(* Schneider Machine Expert - Basic project driveAPIREV3, file version 2.7.0.0 *)
(* ProjectInformations: Name=PlanPAS 2.0 *)

HARDWARE
  Cpu 0: TM221CE16T
  EthernetConfiguration: NetworkName=M221, IpAllocationMode=FixedAddress, IpAddress=192.168.0.2, SubnetMask=255.255.255.0
  SerialLineConfiguration: Baud=Baud19200, Parity=ParityEven, DataBits=DataBits8, StopBits=StopBits1, PhysicalMedium=PhysicalMediumRs485, TransmissionMode=TransmissionModeModbusRtu, SlaveId=1, Addressing=SlaveAddressing
  MastTask: UsePeriodScanMode=false, PeriodScan=100
  FastTask: Period=255
  CpuBehavior: StartingMode=StartAsPreviousState, AutoSaveRamOnEeprom=true, WatchdogPeriod=250

SYMBOLS  (address, symbol, comment, settings)
  %M0         "ESTEIRA"
  %M1         "AVANÇA PISTÃO 1"
  %M2         "AVANÇA PISTÃO 2"
  %M3         "AVANÇA PISTÃO 3"
  %M4         "RETORNA PISTÃO 3"
  %M5         "IDENTIFICA PEÇA NA ESTEIRA (CAPACITIVO)"
  %M6         "LIMPA AVISOS"
  %M10        "MEDIA"
  %M11        "GRANDE"
  %M12        "METAL"
  %M14        "CHEGADA DE PEÇA BOX 2"
  %M15        "CHEGADA DE PEÇA BOX 1"
  %M16        "CHEGADA DE PEÇA BOX 3"
  %M17        "CHEGADA DE PEÇA BOX 4"
  %M20        "PEQ_NMET"
  %M21        "PEQ_MET"
  %M22        "MED_NMET"
  %M23        "MED_MET"
  %M24        "GRD_NMET"
  %M25        "GRD_MET"
  %M30      INICIAR
  %M31      PARAR
  %M32      REPROG
  %M33      VOLTAR
  %M34      INICIADO
  %M40        "INICIAR AUX"
  %M41        "PARAR AUX"
  %M42        "REPROGRAMAR AUX"
  %M43        "VOLTAR AUX"
  %M44        "ZERA MEMORIA SOLICITAÇÕES"
  %MW0        "AVISOS"
  %MW10     CX1MG  "SOLICITAÇÃO"
  %MW11     CX1MM
  %MW12     CX1MP
  %MW13     CX1NMG
  %MW14     CX1NMM
  %MW15     CX1NMP
  %MW16     CX2MG
  %MW17     CX2MM
  %MW18     CX2MP
  %MW19     CX2NMG
  %MW20     CX2NMM
  %MW21     CX2NMP
  %MW22     CX3MG
  %MW23     CX3MM
  %MW24     CX3MP
  %MW25     CX3NMG
  %MW26     CX3NMM
  %MW27     CX3NMP
  %I0.0       "SENS_OTICO_MED"
  %I0.1       "SENS_OTICO_GDE"
  %I0.2       "SENS_INDUTIVO"
  %I0.3       "SENS_CAPACITIVO"
  %I0.4       "FC2"
  %I0.5       "FC1"
  %I0.6       "FC3"
  %I0.7       "FC4"
  %Q0.0       "M1"
  %Q0.1       "AP1"
  %Q0.2       "AP2"
  %Q0.3       "AP3"
  %Q0.5       "RP3"

POU Novo POU
  (* SectionNumber=1 *)

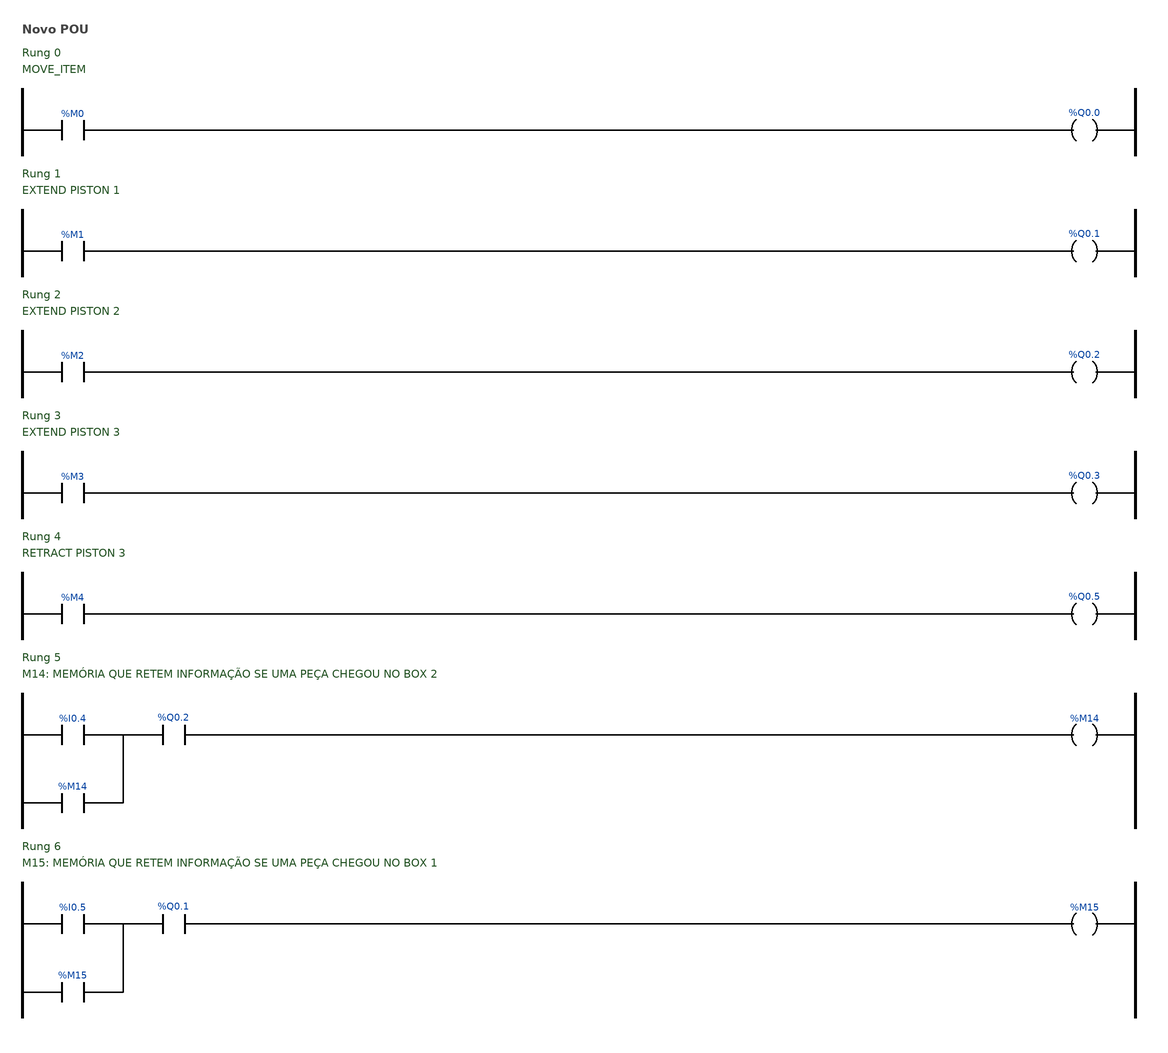

// Rung 0
// MOVE_ITEM
  LD %M0
  ST %Q0.0
  // as ST:
  //   %Q0.0 := %M0;

// Rung 1
// EXTEND PISTON 1
  LD %M1
  ST %Q0.1
  // as ST:
  //   %Q0.1 := %M1;

// Rung 2
// EXTEND PISTON 2
  LD %M2
  ST %Q0.2
  // as ST:
  //   %Q0.2 := %M2;

// Rung 3
// EXTEND PISTON 3
  LD %M3
  ST %Q0.3
  // as ST:
  //   %Q0.3 := %M3;

// Rung 4
// RETRACT PISTON 3
  LD %M4
  ST %Q0.5
  // as ST:
  //   %Q0.5 := %M4;

// Rung 5
// M14: MEMÓRIA QUE RETEM INFORMAÇÃO SE UMA PEÇA CHEGOU NO BOX 2
  LD %I0.4
  OR %M14
  AND %Q0.2
  ST %M14
  // as ST:
  //   %M14 := (%I0.4 OR %M14) AND %Q0.2;

// Rung 6
// M15: MEMÓRIA QUE RETEM INFORMAÇÃO SE UMA PEÇA CHEGOU NO BOX 1
  LD %I0.5
  OR %M15
  AND %Q0.1
  ST %M15
  // as ST:
  //   %M15 := (%I0.5 OR %M15) AND %Q0.1;

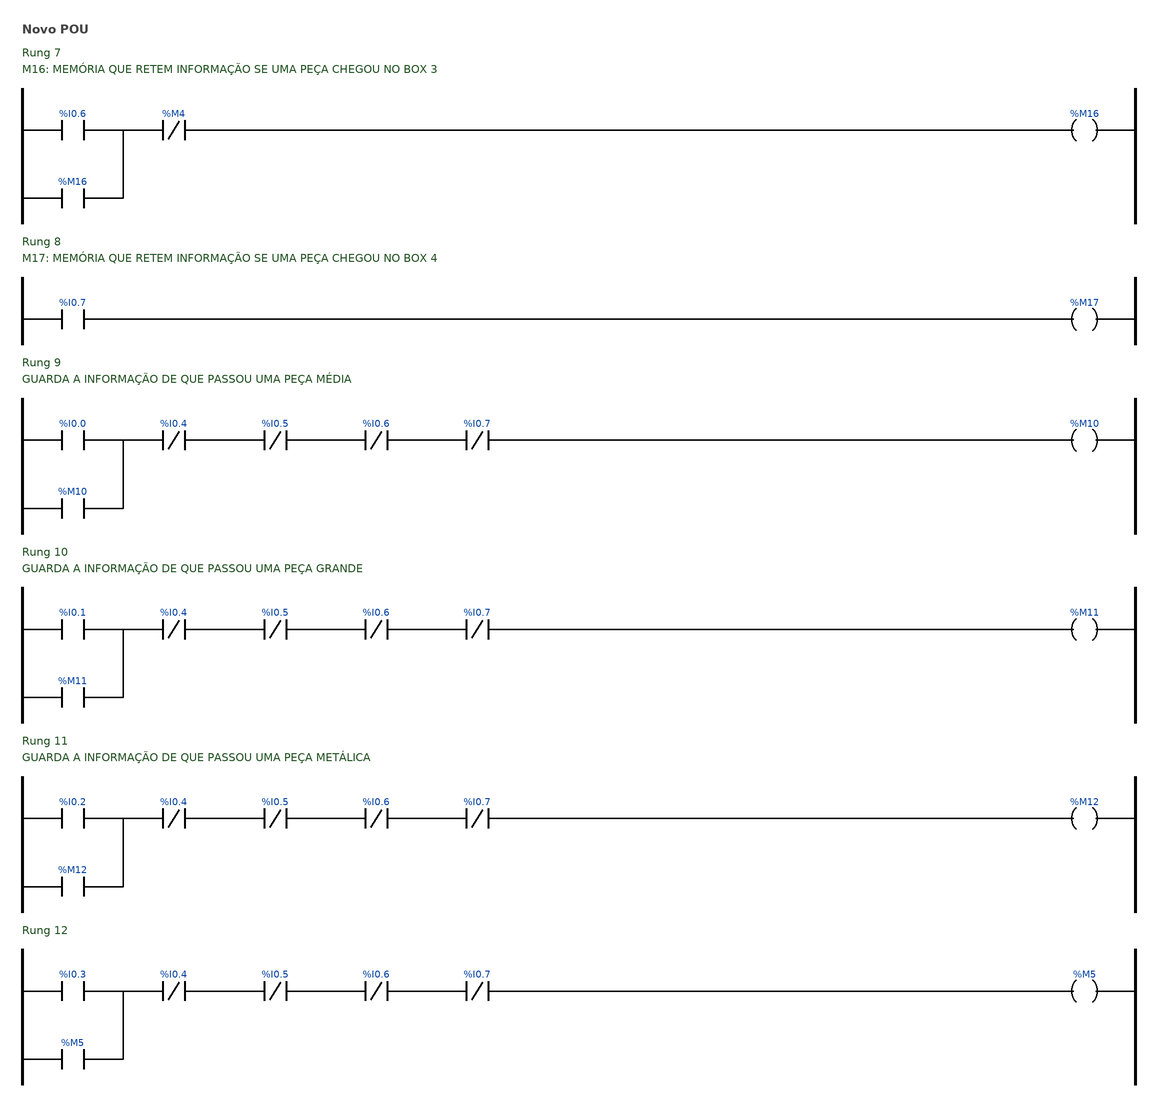

// Rung 7
// M16: MEMÓRIA QUE RETEM INFORMAÇÃO SE UMA PEÇA CHEGOU NO BOX 3
  LD %I0.6
  OR %M16
  ANDN %M4
  ST %M16
  // as ST:
  //   %M16 := (%I0.6 OR %M16) AND NOT %M4;

// Rung 8
// M17: MEMÓRIA QUE RETEM INFORMAÇÃO SE UMA PEÇA CHEGOU NO BOX 4
  LD %I0.7
  ST %M17
  // as ST:
  //   %M17 := %I0.7;

// Rung 9
// GUARDA A INFORMAÇÃO DE QUE PASSOU UMA PEÇA MÉDIA
  LD %I0.0
  OR %M10
  ANDN %I0.4
  ANDN %I0.5
  ANDN %I0.6
  ANDN %I0.7
  ST %M10
  // as ST:
  //   %M10 := (%I0.0 OR %M10) AND NOT %I0.4 AND NOT %I0.5 AND NOT %I0.6 AND NOT %I0.7;

// Rung 10
// GUARDA A INFORMAÇÃO DE QUE PASSOU UMA PEÇA GRANDE
  LD %I0.1
  OR %M11
  ANDN %I0.4
  ANDN %I0.5
  ANDN %I0.6
  ANDN %I0.7
  ST %M11
  // as ST:
  //   %M11 := (%I0.1 OR %M11) AND NOT %I0.4 AND NOT %I0.5 AND NOT %I0.6 AND NOT %I0.7;

// Rung 11
// GUARDA A INFORMAÇÃO DE QUE PASSOU UMA PEÇA METÁLICA
  LD %I0.2
  OR %M12
  ANDN %I0.4
  ANDN %I0.5
  ANDN %I0.6
  ANDN %I0.7
  ST %M12
  // as ST:
  //   %M12 := (%I0.2 OR %M12) AND NOT %I0.4 AND NOT %I0.5 AND NOT %I0.6 AND NOT %I0.7;

// Rung 12
  LD %I0.3
  OR %M5
  ANDN %I0.4
  ANDN %I0.5
  ANDN %I0.6
  ANDN %I0.7
  ST %M5
  // as ST:
  //   %M5 := (%I0.3 OR %M5) AND NOT %I0.4 AND NOT %I0.5 AND NOT %I0.6 AND NOT %I0.7;

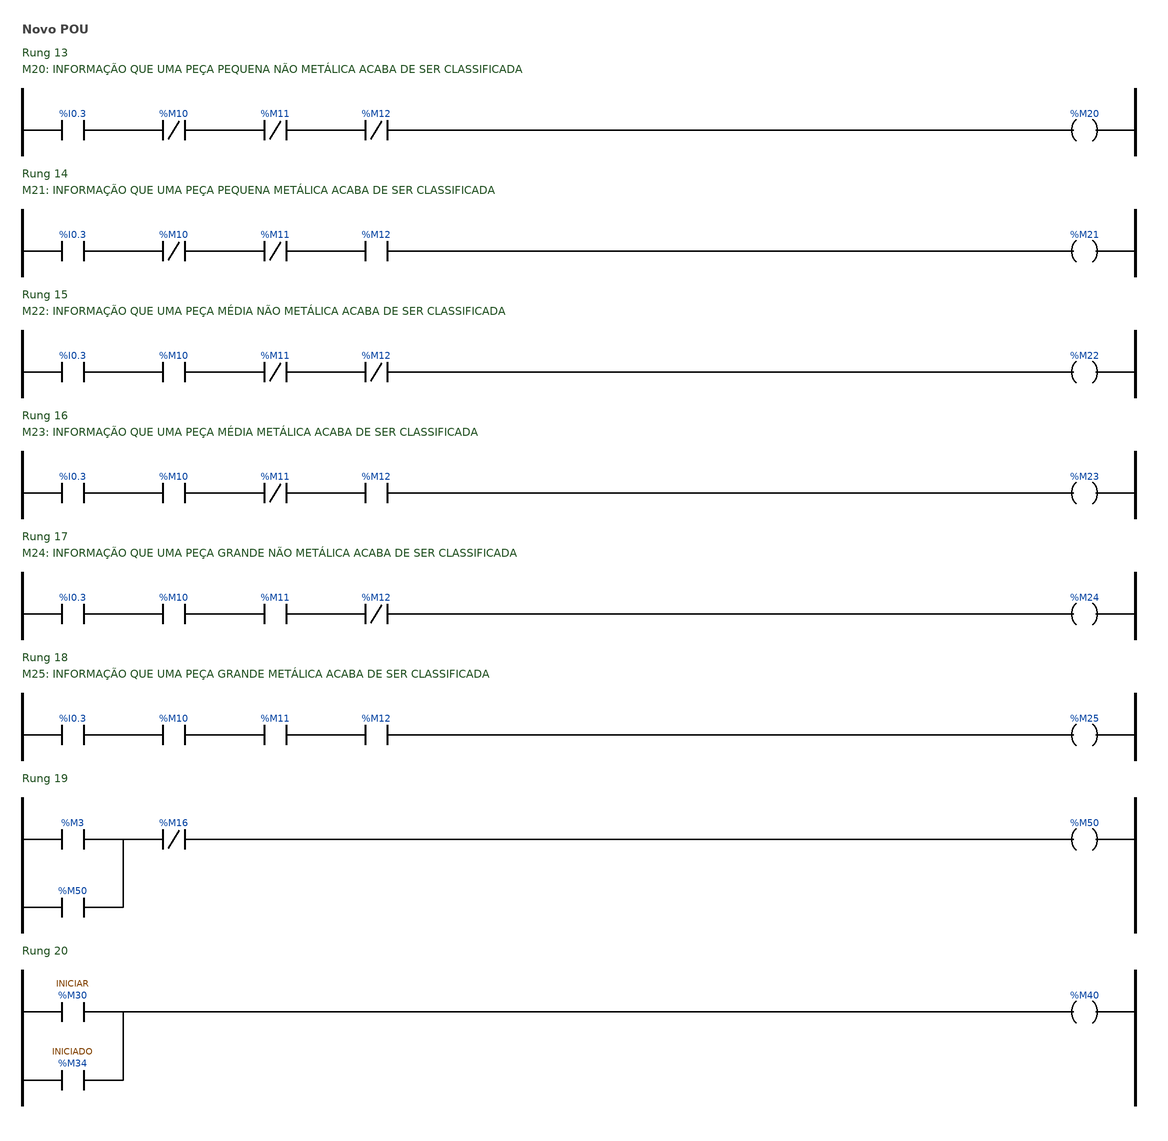

// Rung 13
// M20: INFORMAÇÃO QUE UMA PEÇA PEQUENA NÃO METÁLICA ACABA DE SER CLASSIFICADA
  LD %I0.3
  ANDN %M10
  ANDN %M11
  ANDN %M12
  ST %M20
  // as ST:
  //   %M20 := %I0.3 AND NOT %M10 AND NOT %M11 AND NOT %M12;

// Rung 14
// M21: INFORMAÇÃO QUE UMA PEÇA PEQUENA METÁLICA ACABA DE SER CLASSIFICADA
  LD %I0.3
  ANDN %M10
  ANDN %M11
  AND %M12
  ST %M21
  // as ST:
  //   %M21 := %I0.3 AND NOT %M10 AND NOT %M11 AND %M12;

// Rung 15
// M22: INFORMAÇÃO QUE UMA PEÇA MÉDIA NÃO METÁLICA ACABA DE SER CLASSIFICADA
  LD %I0.3
  AND %M10
  ANDN %M11
  ANDN %M12
  ST %M22
  // as ST:
  //   %M22 := %I0.3 AND %M10 AND NOT %M11 AND NOT %M12;

// Rung 16
// M23: INFORMAÇÃO QUE UMA PEÇA MÉDIA METÁLICA ACABA DE SER CLASSIFICADA
  LD %I0.3
  AND %M10
  ANDN %M11
  AND %M12
  ST %M23
  // as ST:
  //   %M23 := %I0.3 AND %M10 AND NOT %M11 AND %M12;

// Rung 17
// M24: INFORMAÇÃO QUE UMA PEÇA GRANDE NÃO METÁLICA ACABA DE SER CLASSIFICADA
  LD %I0.3
  AND %M10
  AND %M11
  ANDN %M12
  ST %M24
  // as ST:
  //   %M24 := %I0.3 AND %M10 AND %M11 AND NOT %M12;

// Rung 18
// M25: INFORMAÇÃO QUE UMA PEÇA GRANDE METÁLICA ACABA DE SER CLASSIFICADA
  LD %I0.3
  AND %M10
  AND %M11
  AND %M12
  ST %M25
  // as ST:
  //   %M25 := %I0.3 AND %M10 AND %M11 AND %M12;

// Rung 19
  LD %M3
  OR %M50
  ANDN %M16
  ST %M50
  // as ST:
  //   %M50 := (%M3 OR %M50) AND NOT %M16;

// Rung 20
  LD %M30                 (* INICIAR *)
  OR %M34                 (* INICIADO *)
  ST %M40
  // as ST:
  //   %M40 := INICIAR OR INICIADO;

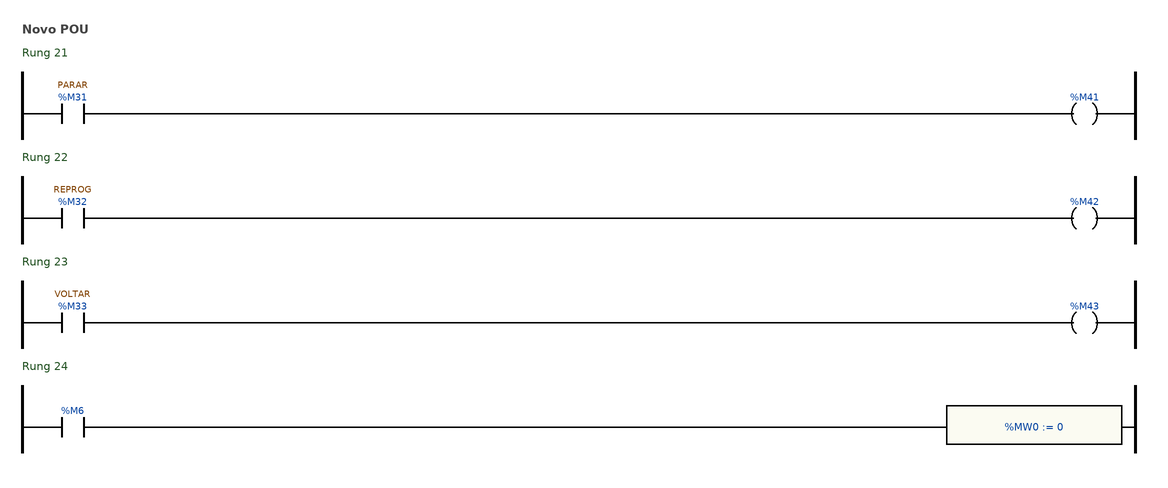

// Rung 21
  LD %M31                 (* PARAR *)
  ST %M41
  // as ST:
  //   %M41 := PARAR;

// Rung 22
  LD %M32                 (* REPROG *)
  ST %M42
  // as ST:
  //   %M42 := REPROG;

// Rung 23
  LD %M33                 (* VOLTAR *)
  ST %M43
  // as ST:
  //   %M43 := VOLTAR;

// Rung 24
  LD %M6
  [ %MW0 := 0 ]
  // as ST:
  //   IF %M6 THEN %MW0 := 0; END_IF;

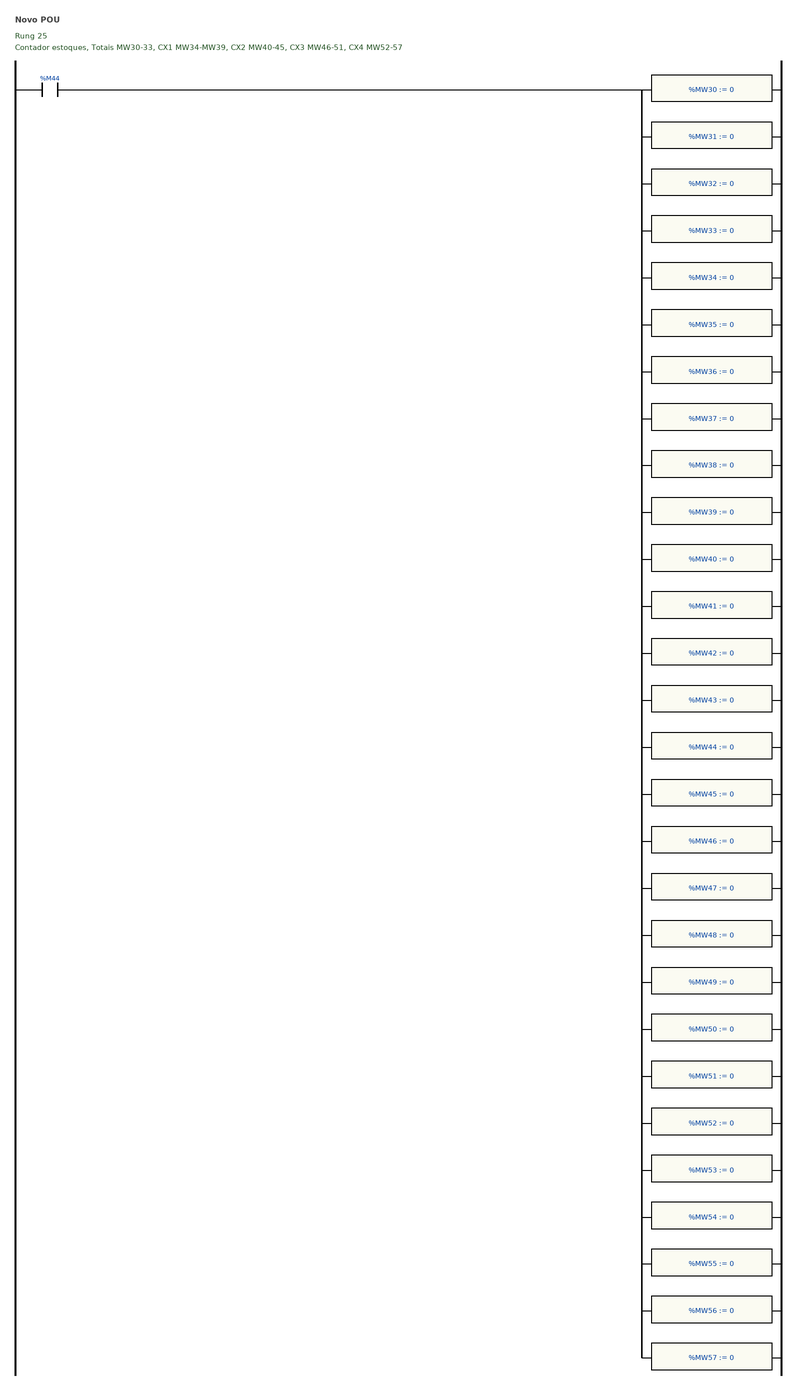

// Rung 25
// Contador estoques, Totais MW30-33, CX1 MW34-MW39, CX2 MW40-45, CX3 MW46-51, CX4 MW52-57
  LD %M44
  [ %MW30 := 0 ]
  [ %MW31 := 0 ]
  [ %MW32 := 0 ]
  [ %MW33 := 0 ]
  [ %MW34 := 0 ]
  [ %MW35 := 0 ]
  [ %MW36 := 0 ]
  [ %MW37 := 0 ]
  [ %MW38 := 0 ]
  [ %MW39 := 0 ]
  [ %MW40 := 0 ]
  [ %MW41 := 0 ]
  [ %MW42 := 0 ]
  [ %MW43 := 0 ]
  [ %MW44 := 0 ]
  [ %MW45 := 0 ]
  [ %MW46 := 0 ]
  [ %MW47 := 0 ]
  [ %MW48 := 0 ]
  [ %MW49 := 0 ]
  [ %MW50 := 0 ]
  [ %MW51 := 0 ]
  [ %MW52 := 0 ]
  [ %MW53 := 0 ]
  [ %MW54 := 0 ]
  [ %MW55 := 0 ]
  [ %MW56 := 0 ]
  [ %MW57 := 0 ]
  // as ST:
  //   IF %M44 THEN %MW30 := 0; END_IF;
  //   IF %M44 THEN %MW31 := 0; END_IF;
  //   IF %M44 THEN %MW32 := 0; END_IF;
  //   IF %M44 THEN %MW33 := 0; END_IF;
  //   IF %M44 THEN %MW34 := 0; END_IF;
  //   IF %M44 THEN %MW35 := 0; END_IF;
  //   IF %M44 THEN %MW36 := 0; END_IF;
  //   IF %M44 THEN %MW37 := 0; END_IF;
  //   IF %M44 THEN %MW38 := 0; END_IF;
  //   IF %M44 THEN %MW39 := 0; END_IF;
  //   IF %M44 THEN %MW40 := 0; END_IF;
  //   IF %M44 THEN %MW41 := 0; END_IF;
  //   IF %M44 THEN %MW42 := 0; END_IF;
  //   IF %M44 THEN %MW43 := 0; END_IF;
  //   IF %M44 THEN %MW44 := 0; END_IF;
  //   IF %M44 THEN %MW45 := 0; END_IF;
  //   IF %M44 THEN %MW46 := 0; END_IF;
  //   IF %M44 THEN %MW47 := 0; END_IF;
  //   IF %M44 THEN %MW48 := 0; END_IF;
  //   IF %M44 THEN %MW49 := 0; END_IF;
  //   IF %M44 THEN %MW50 := 0; END_IF;
  //   IF %M44 THEN %MW51 := 0; END_IF;
  //   IF %M44 THEN %MW52 := 0; END_IF;
  //   IF %M44 THEN %MW53 := 0; END_IF;
  //   IF %M44 THEN %MW54 := 0; END_IF;
  //   IF %M44 THEN %MW55 := 0; END_IF;
  //   IF %M44 THEN %MW56 := 0; END_IF;
  //   IF %M44 THEN %MW57 := 0; END_IF;

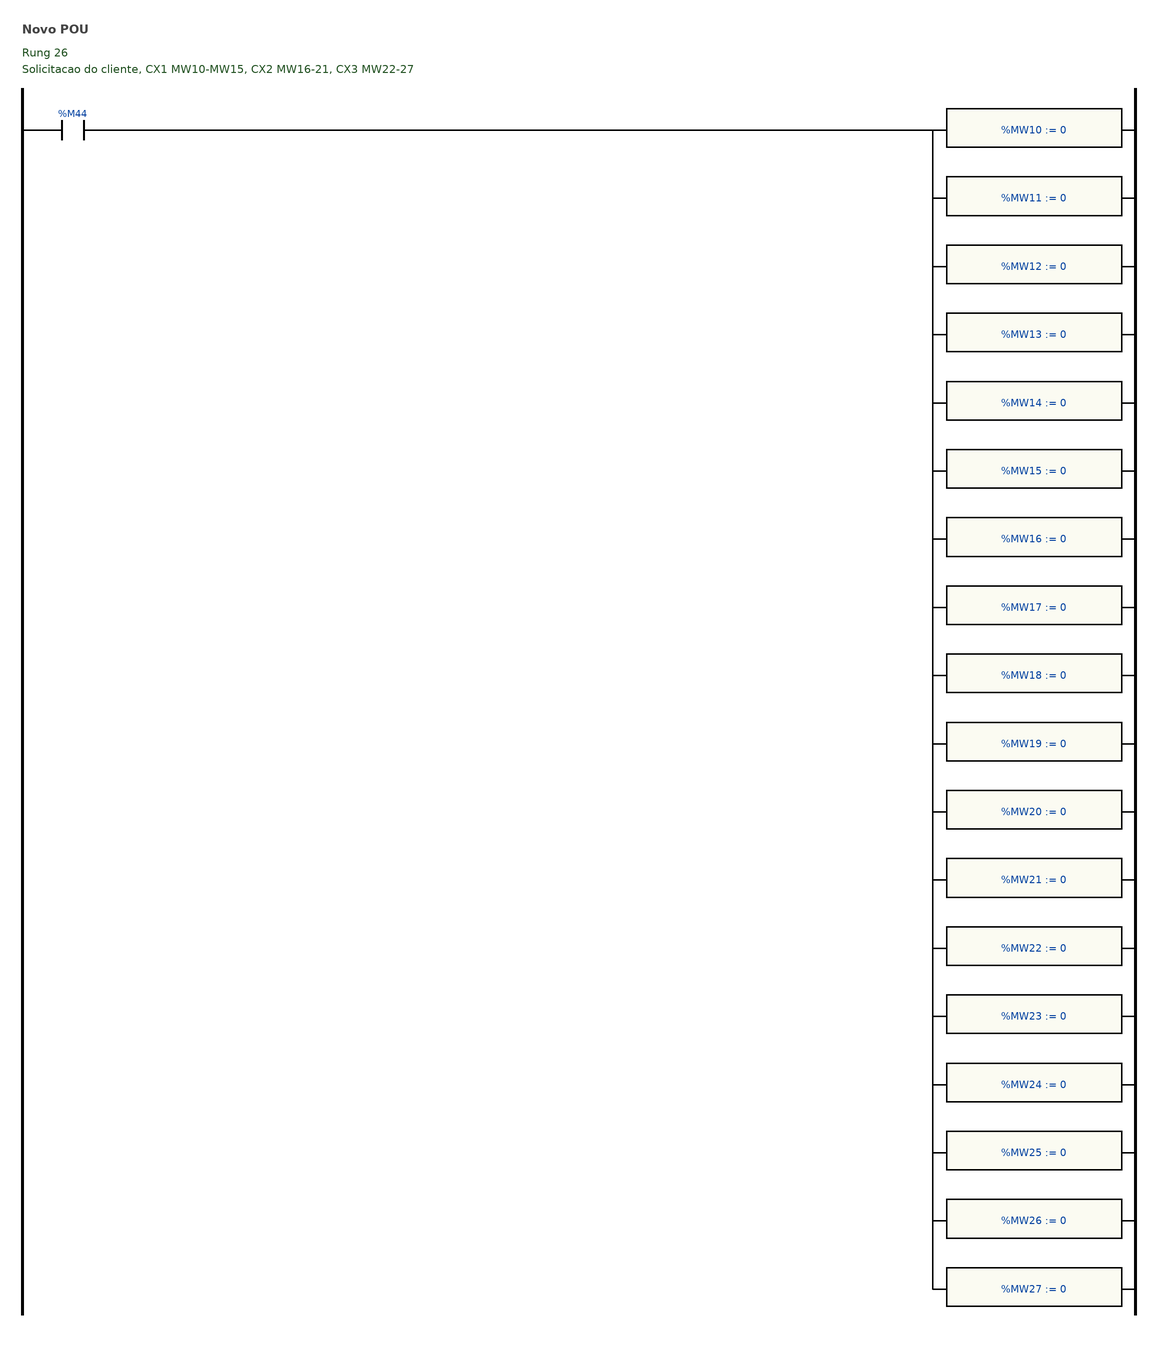

// Rung 26
// Solicitacao do cliente, CX1 MW10-MW15, CX2 MW16-21, CX3 MW22-27
  LD %M44
  [ %MW10 := 0 ]          (* CX1MG *)
  [ %MW11 := 0 ]          (* CX1MM *)
  [ %MW12 := 0 ]          (* CX1MP *)
  [ %MW13 := 0 ]          (* CX1NMG *)
  [ %MW14 := 0 ]          (* CX1NMM *)
  [ %MW15 := 0 ]          (* CX1NMP *)
  [ %MW16 := 0 ]          (* CX2MG *)
  [ %MW17 := 0 ]          (* CX2MM *)
  [ %MW18 := 0 ]          (* CX2MP *)
  [ %MW19 := 0 ]          (* CX2NMG *)
  [ %MW20 := 0 ]          (* CX2NMM *)
  [ %MW21 := 0 ]          (* CX2NMP *)
  [ %MW22 := 0 ]          (* CX3MG *)
  [ %MW23 := 0 ]          (* CX3MM *)
  [ %MW24 := 0 ]          (* CX3MP *)
  [ %MW25 := 0 ]          (* CX3NMG *)
  [ %MW26 := 0 ]          (* CX3NMM *)
  [ %MW27 := 0 ]          (* CX3NMP *)
  // as ST:
  //   IF %M44 THEN CX1MG := 0; END_IF;
  //   IF %M44 THEN CX1MM := 0; END_IF;
  //   IF %M44 THEN CX1MP := 0; END_IF;
  //   IF %M44 THEN CX1NMG := 0; END_IF;
  //   IF %M44 THEN CX1NMM := 0; END_IF;
  //   IF %M44 THEN CX1NMP := 0; END_IF;
  //   IF %M44 THEN CX2MG := 0; END_IF;
  //   IF %M44 THEN CX2MM := 0; END_IF;
  //   IF %M44 THEN CX2MP := 0; END_IF;
  //   IF %M44 THEN CX2NMG := 0; END_IF;
  //   IF %M44 THEN CX2NMM := 0; END_IF;
  //   IF %M44 THEN CX2NMP := 0; END_IF;
  //   IF %M44 THEN CX3MG := 0; END_IF;
  //   IF %M44 THEN CX3MM := 0; END_IF;
  //   IF %M44 THEN CX3MP := 0; END_IF;
  //   IF %M44 THEN CX3NMG := 0; END_IF;
  //   IF %M44 THEN CX3NMM := 0; END_IF;
  //   IF %M44 THEN CX3NMP := 0; END_IF;
